// TIA Portal V17 export
// export: Created 2023-04-03T06:31:36.8753928Z, ExportSetting WithDefaults, DisplayName Totally Integrated Automation Portal, DisplayVersion V17 Update 4, DisplayName TIA Portal Openness, DisplayVersion V17 Update 4, DisplayName TIA Portal Version Control Interface, DisplayVersion V17, DisplayName STEP 7 Professional, DisplayVersion V17 Update 4, DisplayName STEP 7 Safety, DisplayVersion V17, DisplayName WinCC Professional, DisplayVersion V17 Update 4
ORGANIZATION_BLOCK "Main"   // OB1, LAD, ProgramCycle
TITLE = "Main Program Sweep (Cycle)"
{ S7_Optimized_Access := 'TRUE' }
VERSION : 0.1
// stored: AutoNumber true, IsIECCheckEnabled false, SetENOAutomatically false
   VAR_INPUT
      Initial_Call : Bool;   // Initial call of this OB
      Remanence : Bool;   // =True, if remanent data are available
   END_VAR
BEGIN

REGION Network 1: Acknowledgement ProfiSafe
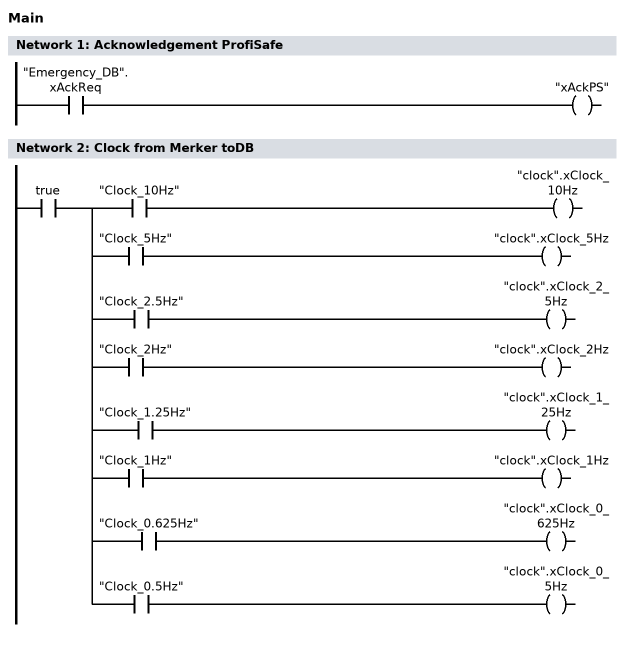
   RUNG wire#powerrail
      Contact( "Emergency_DB".xAckReq )
      Coil( "xAckPS" )
   END_RUNG
   // the same network as SCL:
   "xAckPS" := "Emergency_DB".xAckReq;
END_REGION

REGION Network 2: Clock from Merker toDB
   RUNG wire#powerrail
      Contact( true )
      wire#w1
      Contact( "Clock_10Hz" )
      Coil( "clock".xClock_10Hz )
   END_RUNG
   RUNG wire#w1
      Contact( "Clock_5Hz" )
      Coil( "clock".xClock_5Hz )
   END_RUNG
   RUNG wire#w1
      Contact( "Clock_2.5Hz" )
      Coil( "clock".xClock_2_5Hz )
   END_RUNG
   RUNG wire#w1
      Contact( "Clock_2Hz" )
      Coil( "clock".xClock_2Hz )
   END_RUNG
   RUNG wire#w1
      Contact( "Clock_1.25Hz" )
      Coil( "clock".xClock_1_25Hz )
   END_RUNG
   RUNG wire#w1
      Contact( "Clock_1Hz" )
      Coil( "clock".xClock_1Hz )
   END_RUNG
   RUNG wire#w1
      Contact( "Clock_0.625Hz" )
      Coil( "clock".xClock_0_625Hz )
   END_RUNG
   RUNG wire#w1
      Contact( "Clock_0.5Hz" )
      Coil( "clock".xClock_0_5Hz )
   END_RUNG
   // the same network as SCL:
   "clock".xClock_10Hz := true AND "Clock_10Hz";
   "clock".xClock_5Hz := true AND "Clock_5Hz";
   "clock".xClock_2_5Hz := true AND "Clock_2.5Hz";
   "clock".xClock_2Hz := true AND "Clock_2Hz";
   "clock".xClock_1_25Hz := true AND "Clock_1.25Hz";
   "clock".xClock_1Hz := true AND "Clock_1Hz";
   "clock".xClock_0_625Hz := true AND "Clock_0.625Hz";
   "clock".xClock_0_5Hz := true AND "Clock_0.5Hz";
END_REGION
END_ORGANIZATION_BLOCK
